FUNCTION_BLOCK Testowy2
VAR
	bTest: BOOL;
END_VAR

END_FUNCTION_BLOCK

(* stored: Version 1.1.0.1
   POU Testowy2: Id {84d8b5d7-d81e-4100-ad6d-92aa37f81770}, SpecialFunc None *)
